// TIA Portal V15.1 export
// export: Created 2022-12-22T12:03:23.8131243Z, ExportSetting None, DisplayName Totally Integrated Automation Portal, DisplayVersion V15.1 Update 5, DisplayName TIA Portal Openness, DisplayVersion V15.1 Update 5, DisplayName TIA Portal Teamcenter Gateway, DisplayVersion V15.1 Update 5, DisplayName SINAMICS Startdrive Advanced, DisplayVersion V15.1, DisplayName G130, G150, S120, S150, SINAMICS MV, S210, DisplayVersion V15.1, DisplayName G110M, G120, G120C, G120D, G120P, DisplayVersion V15.1, DisplayName STEP 7 Professional, DisplayVersion V15.1 Update 5, DisplayName Soft Starter ES, DisplayVersion V15.1, DisplayName WinCC Professional, DisplayVersion V15.1 Update 5, DisplayName SIMATIC Visualization Architect, DisplayVersion V15.1
FUNCTION "CallTemplate" : Void   // FC10, LAD
{ S7_Optimized_Access := 'TRUE' }
// stored: SetENOAutomatically False
   VAR_TEMP
      t_PowerRelease : Bool;
   END_VAR
BEGIN

REGION Network 1: Release by power
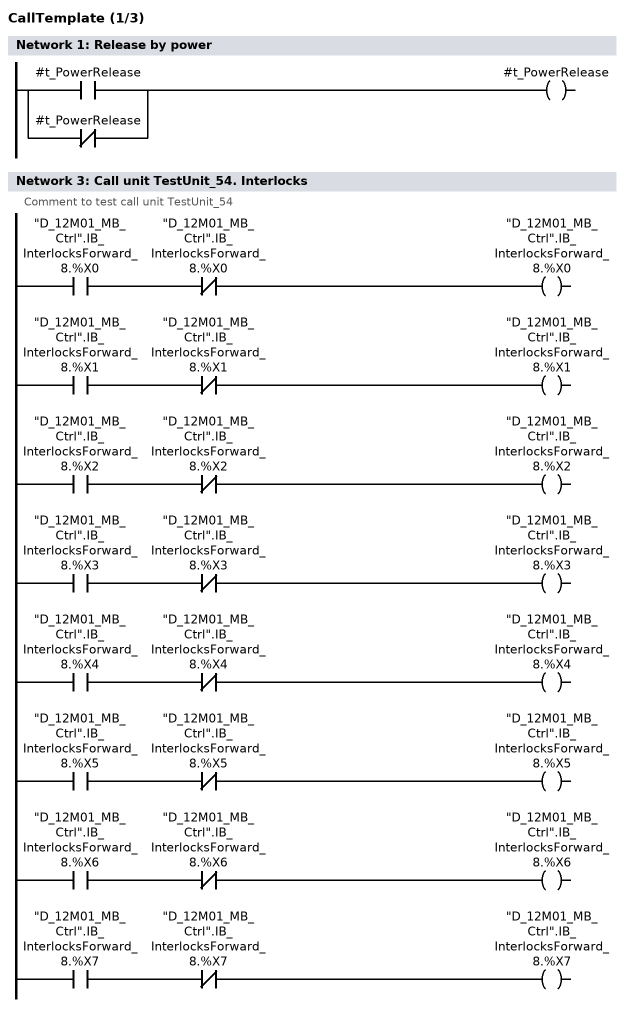
   RUNG wire#powerrail
      Contact( #t_PowerRelease )
      wire#w1
      Coil( #t_PowerRelease )
   END_RUNG
   RUNG wire#powerrail
      I_Contact( #t_PowerRelease )
   END_RUNG wire#w1
   // the same network as SCL:
   #t_PowerRelease := #t_PowerRelease OR NOT #t_PowerRelease;
END_REGION

REGION Network 3: Call unit TestUnit_54. Interlocks
   // Comment to test call unit TestUnit_54
   RUNG wire#powerrail
      Contact( "D_12M01_MB_Ctrl".IB_InterlocksForward_8.%X0 )
      I_Contact( "D_12M01_MB_Ctrl".IB_InterlocksForward_8.%X0 )
      Coil( "D_12M01_MB_Ctrl".IB_InterlocksForward_8.%X0 )
   END_RUNG
   RUNG wire#powerrail
      Contact( "D_12M01_MB_Ctrl".IB_InterlocksForward_8.%X1 )
      I_Contact( "D_12M01_MB_Ctrl".IB_InterlocksForward_8.%X1 )
      Coil( "D_12M01_MB_Ctrl".IB_InterlocksForward_8.%X1 )
   END_RUNG
   RUNG wire#powerrail
      Contact( "D_12M01_MB_Ctrl".IB_InterlocksForward_8.%X2 )
      I_Contact( "D_12M01_MB_Ctrl".IB_InterlocksForward_8.%X2 )
      Coil( "D_12M01_MB_Ctrl".IB_InterlocksForward_8.%X2 )
   END_RUNG
   RUNG wire#powerrail
      Contact( "D_12M01_MB_Ctrl".IB_InterlocksForward_8.%X3 )
      I_Contact( "D_12M01_MB_Ctrl".IB_InterlocksForward_8.%X3 )
      Coil( "D_12M01_MB_Ctrl".IB_InterlocksForward_8.%X3 )
   END_RUNG
   RUNG wire#powerrail
      Contact( "D_12M01_MB_Ctrl".IB_InterlocksForward_8.%X4 )
      I_Contact( "D_12M01_MB_Ctrl".IB_InterlocksForward_8.%X4 )
      Coil( "D_12M01_MB_Ctrl".IB_InterlocksForward_8.%X4 )
   END_RUNG
   RUNG wire#powerrail
      Contact( "D_12M01_MB_Ctrl".IB_InterlocksForward_8.%X5 )
      I_Contact( "D_12M01_MB_Ctrl".IB_InterlocksForward_8.%X5 )
      Coil( "D_12M01_MB_Ctrl".IB_InterlocksForward_8.%X5 )
   END_RUNG
   RUNG wire#powerrail
      Contact( "D_12M01_MB_Ctrl".IB_InterlocksForward_8.%X6 )
      I_Contact( "D_12M01_MB_Ctrl".IB_InterlocksForward_8.%X6 )
      Coil( "D_12M01_MB_Ctrl".IB_InterlocksForward_8.%X6 )
   END_RUNG
   RUNG wire#powerrail
      Contact( "D_12M01_MB_Ctrl".IB_InterlocksForward_8.%X7 )
      I_Contact( "D_12M01_MB_Ctrl".IB_InterlocksForward_8.%X7 )
      Coil( "D_12M01_MB_Ctrl".IB_InterlocksForward_8.%X7 )
   END_RUNG
   // the same network as SCL:
   "D_12M01_MB_Ctrl".IB_InterlocksForward_8.%X0 := "D_12M01_MB_Ctrl".IB_InterlocksForward_8.%X0 AND NOT "D_12M01_MB_Ctrl".IB_InterlocksForward_8.%X0;
   "D_12M01_MB_Ctrl".IB_InterlocksForward_8.%X1 := "D_12M01_MB_Ctrl".IB_InterlocksForward_8.%X1 AND NOT "D_12M01_MB_Ctrl".IB_InterlocksForward_8.%X1;
   "D_12M01_MB_Ctrl".IB_InterlocksForward_8.%X2 := "D_12M01_MB_Ctrl".IB_InterlocksForward_8.%X2 AND NOT "D_12M01_MB_Ctrl".IB_InterlocksForward_8.%X2;
   "D_12M01_MB_Ctrl".IB_InterlocksForward_8.%X3 := "D_12M01_MB_Ctrl".IB_InterlocksForward_8.%X3 AND NOT "D_12M01_MB_Ctrl".IB_InterlocksForward_8.%X3;
   "D_12M01_MB_Ctrl".IB_InterlocksForward_8.%X4 := "D_12M01_MB_Ctrl".IB_InterlocksForward_8.%X4 AND NOT "D_12M01_MB_Ctrl".IB_InterlocksForward_8.%X4;
   "D_12M01_MB_Ctrl".IB_InterlocksForward_8.%X5 := "D_12M01_MB_Ctrl".IB_InterlocksForward_8.%X5 AND NOT "D_12M01_MB_Ctrl".IB_InterlocksForward_8.%X5;
   "D_12M01_MB_Ctrl".IB_InterlocksForward_8.%X6 := "D_12M01_MB_Ctrl".IB_InterlocksForward_8.%X6 AND NOT "D_12M01_MB_Ctrl".IB_InterlocksForward_8.%X6;
   "D_12M01_MB_Ctrl".IB_InterlocksForward_8.%X7 := "D_12M01_MB_Ctrl".IB_InterlocksForward_8.%X7 AND NOT "D_12M01_MB_Ctrl".IB_InterlocksForward_8.%X7;
END_REGION

REGION Network 4: Call unit TestUnit_54. External faults
   // Comment to test call unit TestUnit_54
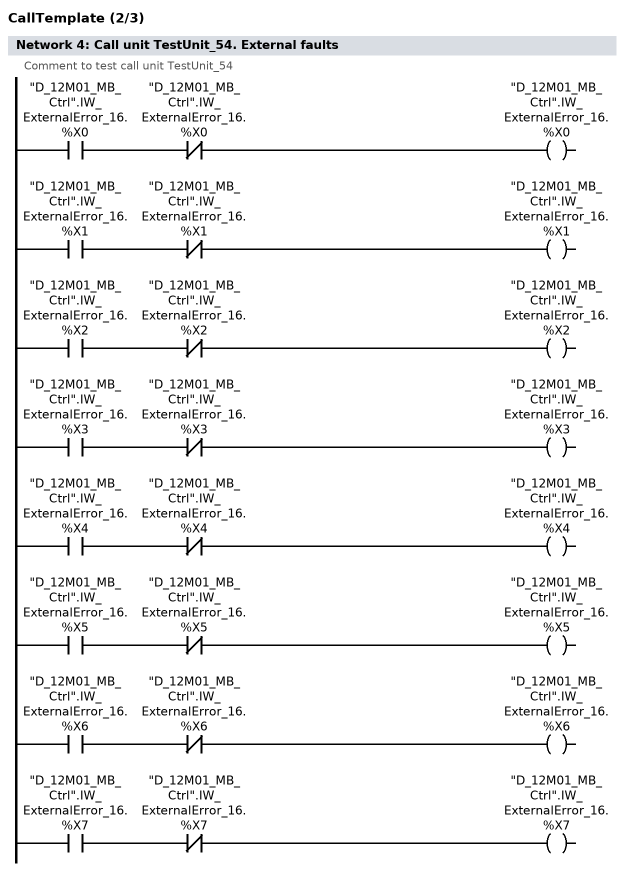
   RUNG wire#powerrail
      Contact( "D_12M01_MB_Ctrl".IW_ExternalError_16.%X0 )
      I_Contact( "D_12M01_MB_Ctrl".IW_ExternalError_16.%X0 )
      Coil( "D_12M01_MB_Ctrl".IW_ExternalError_16.%X0 )
   END_RUNG
   RUNG wire#powerrail
      Contact( "D_12M01_MB_Ctrl".IW_ExternalError_16.%X1 )
      I_Contact( "D_12M01_MB_Ctrl".IW_ExternalError_16.%X1 )
      Coil( "D_12M01_MB_Ctrl".IW_ExternalError_16.%X1 )
   END_RUNG
   RUNG wire#powerrail
      Contact( "D_12M01_MB_Ctrl".IW_ExternalError_16.%X2 )
      I_Contact( "D_12M01_MB_Ctrl".IW_ExternalError_16.%X2 )
      Coil( "D_12M01_MB_Ctrl".IW_ExternalError_16.%X2 )
   END_RUNG
   RUNG wire#powerrail
      Contact( "D_12M01_MB_Ctrl".IW_ExternalError_16.%X3 )
      I_Contact( "D_12M01_MB_Ctrl".IW_ExternalError_16.%X3 )
      Coil( "D_12M01_MB_Ctrl".IW_ExternalError_16.%X3 )
   END_RUNG
   RUNG wire#powerrail
      Contact( "D_12M01_MB_Ctrl".IW_ExternalError_16.%X4 )
      I_Contact( "D_12M01_MB_Ctrl".IW_ExternalError_16.%X4 )
      Coil( "D_12M01_MB_Ctrl".IW_ExternalError_16.%X4 )
   END_RUNG
   RUNG wire#powerrail
      Contact( "D_12M01_MB_Ctrl".IW_ExternalError_16.%X5 )
      I_Contact( "D_12M01_MB_Ctrl".IW_ExternalError_16.%X5 )
      Coil( "D_12M01_MB_Ctrl".IW_ExternalError_16.%X5 )
   END_RUNG
   RUNG wire#powerrail
      Contact( "D_12M01_MB_Ctrl".IW_ExternalError_16.%X6 )
      I_Contact( "D_12M01_MB_Ctrl".IW_ExternalError_16.%X6 )
      Coil( "D_12M01_MB_Ctrl".IW_ExternalError_16.%X6 )
   END_RUNG
   RUNG wire#powerrail
      Contact( "D_12M01_MB_Ctrl".IW_ExternalError_16.%X7 )
      I_Contact( "D_12M01_MB_Ctrl".IW_ExternalError_16.%X7 )
      Coil( "D_12M01_MB_Ctrl".IW_ExternalError_16.%X7 )
   END_RUNG
   // the same network as SCL:
   "D_12M01_MB_Ctrl".IW_ExternalError_16.%X0 := "D_12M01_MB_Ctrl".IW_ExternalError_16.%X0 AND NOT "D_12M01_MB_Ctrl".IW_ExternalError_16.%X0;
   "D_12M01_MB_Ctrl".IW_ExternalError_16.%X1 := "D_12M01_MB_Ctrl".IW_ExternalError_16.%X1 AND NOT "D_12M01_MB_Ctrl".IW_ExternalError_16.%X1;
   "D_12M01_MB_Ctrl".IW_ExternalError_16.%X2 := "D_12M01_MB_Ctrl".IW_ExternalError_16.%X2 AND NOT "D_12M01_MB_Ctrl".IW_ExternalError_16.%X2;
   "D_12M01_MB_Ctrl".IW_ExternalError_16.%X3 := "D_12M01_MB_Ctrl".IW_ExternalError_16.%X3 AND NOT "D_12M01_MB_Ctrl".IW_ExternalError_16.%X3;
   "D_12M01_MB_Ctrl".IW_ExternalError_16.%X4 := "D_12M01_MB_Ctrl".IW_ExternalError_16.%X4 AND NOT "D_12M01_MB_Ctrl".IW_ExternalError_16.%X4;
   "D_12M01_MB_Ctrl".IW_ExternalError_16.%X5 := "D_12M01_MB_Ctrl".IW_ExternalError_16.%X5 AND NOT "D_12M01_MB_Ctrl".IW_ExternalError_16.%X5;
   "D_12M01_MB_Ctrl".IW_ExternalError_16.%X6 := "D_12M01_MB_Ctrl".IW_ExternalError_16.%X6 AND NOT "D_12M01_MB_Ctrl".IW_ExternalError_16.%X6;
   "D_12M01_MB_Ctrl".IW_ExternalError_16.%X7 := "D_12M01_MB_Ctrl".IW_ExternalError_16.%X7 AND NOT "D_12M01_MB_Ctrl".IW_ExternalError_16.%X7;
END_REGION

REGION Network 5: Call unit TestUnit_54. Control block
   // Comment to test call unit TestUnit_54
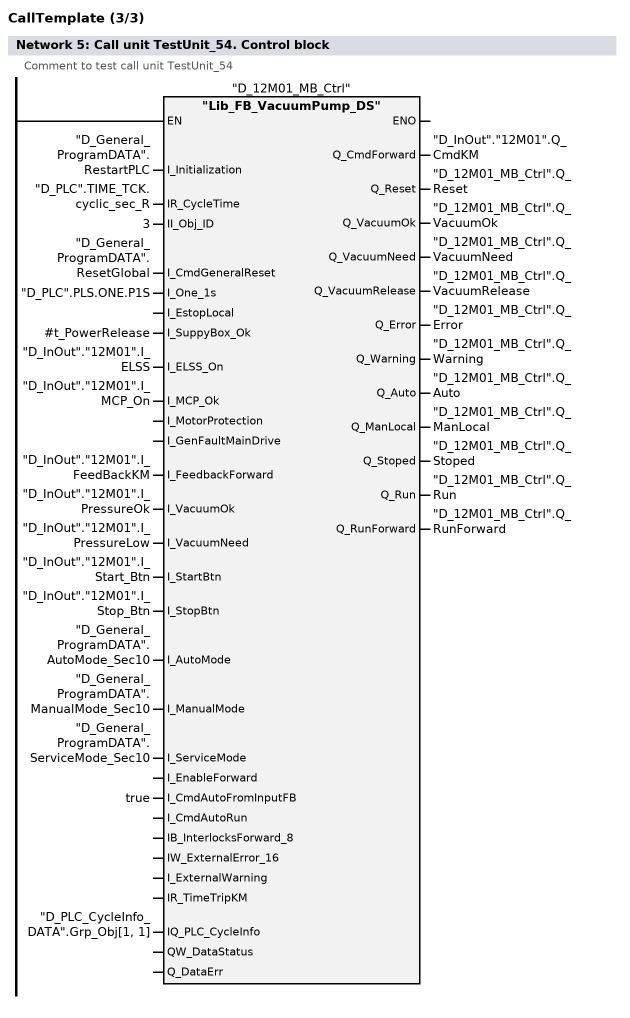
   RUNG wire#powerrail
      "D_12M01_MB_Ctrl"(I_Initialization := "D_General_ProgramDATA".RestartPLC, IR_CycleTime := "D_PLC".TIME_TCK.cyclic_sec_R, II_Obj_ID := 3, I_CmdGeneralReset := "D_General_ProgramDATA".ResetGlobal, I_One_1s := "D_PLC".PLS.ONE.P1S, I_EstopLocal :=, I_SuppyBox_Ok := #t_PowerRelease, I_ELSS_On := "D_InOut"."12M01".I_ELSS, I_MCP_Ok := "D_InOut"."12M01".I_MCP_On, I_MotorProtection :=, I_GenFaultMainDrive :=, I_FeedbackForward := "D_InOut"."12M01".I_FeedBackKM, I_VacuumOk := "D_InOut"."12M01".I_PressureOk, I_VacuumNeed := "D_InOut"."12M01".I_PressureLow, I_StartBtn := "D_InOut"."12M01".I_Start_Btn, I_StopBtn := "D_InOut"."12M01".I_Stop_Btn, I_AutoMode := "D_General_ProgramDATA".AutoMode_Sec10, I_ManualMode := "D_General_ProgramDATA".ManualMode_Sec10, I_ServiceMode := "D_General_ProgramDATA".ServiceMode_Sec10, I_EnableForward :=, I_CmdAutoFromInputFB := true, I_CmdAutoRun :=, IB_InterlocksForward_8 :=, IW_ExternalError_16 :=, I_ExternalWarning :=, IR_TimeTripKM :=, IQ_PLC_CycleInfo := "D_PLC_CycleInfo_DATA".Grp_Obj[1, 1], QW_DataStatus :=, Q_DataErr :=, Q_CmdForward => "D_InOut"."12M01".Q_CmdKM, Q_Reset => "D_12M01_MB_Ctrl".Q_Reset, Q_VacuumOk => "D_12M01_MB_Ctrl".Q_VacuumOk, Q_VacuumNeed => "D_12M01_MB_Ctrl".Q_VacuumNeed, Q_VacuumRelease => "D_12M01_MB_Ctrl".Q_VacuumRelease, Q_Error => "D_12M01_MB_Ctrl".Q_Error, Q_Warning => "D_12M01_MB_Ctrl".Q_Warning, Q_Auto => "D_12M01_MB_Ctrl".Q_Auto, Q_ManLocal => "D_12M01_MB_Ctrl".Q_ManLocal, Q_Stoped => "D_12M01_MB_Ctrl".Q_Stoped, Q_Run => "D_12M01_MB_Ctrl".Q_Run, Q_RunForward => "D_12M01_MB_Ctrl".Q_RunForward)
   END_RUNG
   // the same network as SCL:
   "D_12M01_MB_Ctrl"(I_Initialization := "D_General_ProgramDATA".RestartPLC,   // "Lib_FB_VacuumPump_DS"
                     IR_CycleTime := "D_PLC".TIME_TCK.cyclic_sec_R,
                     II_Obj_ID := 3,
                     I_CmdGeneralReset := "D_General_ProgramDATA".ResetGlobal,
                     I_One_1s := "D_PLC".PLS.ONE.P1S,
                     I_SuppyBox_Ok := #t_PowerRelease,
                     I_ELSS_On := "D_InOut"."12M01".I_ELSS,
                     I_MCP_Ok := "D_InOut"."12M01".I_MCP_On,
                     I_FeedbackForward := "D_InOut"."12M01".I_FeedBackKM,
                     I_VacuumOk := "D_InOut"."12M01".I_PressureOk,
                     I_VacuumNeed := "D_InOut"."12M01".I_PressureLow,
                     I_StartBtn := "D_InOut"."12M01".I_Start_Btn,
                     I_StopBtn := "D_InOut"."12M01".I_Stop_Btn,
                     I_AutoMode := "D_General_ProgramDATA".AutoMode_Sec10,
                     I_ManualMode := "D_General_ProgramDATA".ManualMode_Sec10,
                     I_ServiceMode := "D_General_ProgramDATA".ServiceMode_Sec10,
                     I_CmdAutoFromInputFB := true,
                     IQ_PLC_CycleInfo := "D_PLC_CycleInfo_DATA".Grp_Obj[1, 1],
                     Q_CmdForward => "D_InOut"."12M01".Q_CmdKM,
                     Q_Reset => "D_12M01_MB_Ctrl".Q_Reset,
                     Q_VacuumOk => "D_12M01_MB_Ctrl".Q_VacuumOk,
                     Q_VacuumNeed => "D_12M01_MB_Ctrl".Q_VacuumNeed,
                     Q_VacuumRelease => "D_12M01_MB_Ctrl".Q_VacuumRelease,
                     Q_Error => "D_12M01_MB_Ctrl".Q_Error,
                     Q_Warning => "D_12M01_MB_Ctrl".Q_Warning,
                     Q_Auto => "D_12M01_MB_Ctrl".Q_Auto,
                     Q_ManLocal => "D_12M01_MB_Ctrl".Q_ManLocal,
                     Q_Stoped => "D_12M01_MB_Ctrl".Q_Stoped,
                     Q_Run => "D_12M01_MB_Ctrl".Q_Run,
                     Q_RunForward => "D_12M01_MB_Ctrl".Q_RunForward);
END_REGION
END_FUNCTION
